SYSTEM Test_10 (* System Configuration *)
  (* Standard: 61499-1 *)
  (* Version 0.3, 2003-12-05, JHC, Rockwell Automation, Renamed from NEWSYSTEM. *)
  (* Version 0.2, 2002-11-05, JHC, Rockwell Automation, Fixed missing (empty) FBD in Application. *)
  (* Version 0.1, 2002-01-17, JHC, Rockwell Automation, Minor cleanup *)
  (* Version 0.0, 2000-05-27, JHC, Rockwell Automation *)
  APPLICATION APP1
  END_APPLICATION
  DEVICE HMI : FRAME_DEVICE(BOUNDS := [500,300,700,500], GRID := [1,1])
    RESOURCE Worker1 : PANEL_RESOURCE(ROWS := 4, COLS := 2)
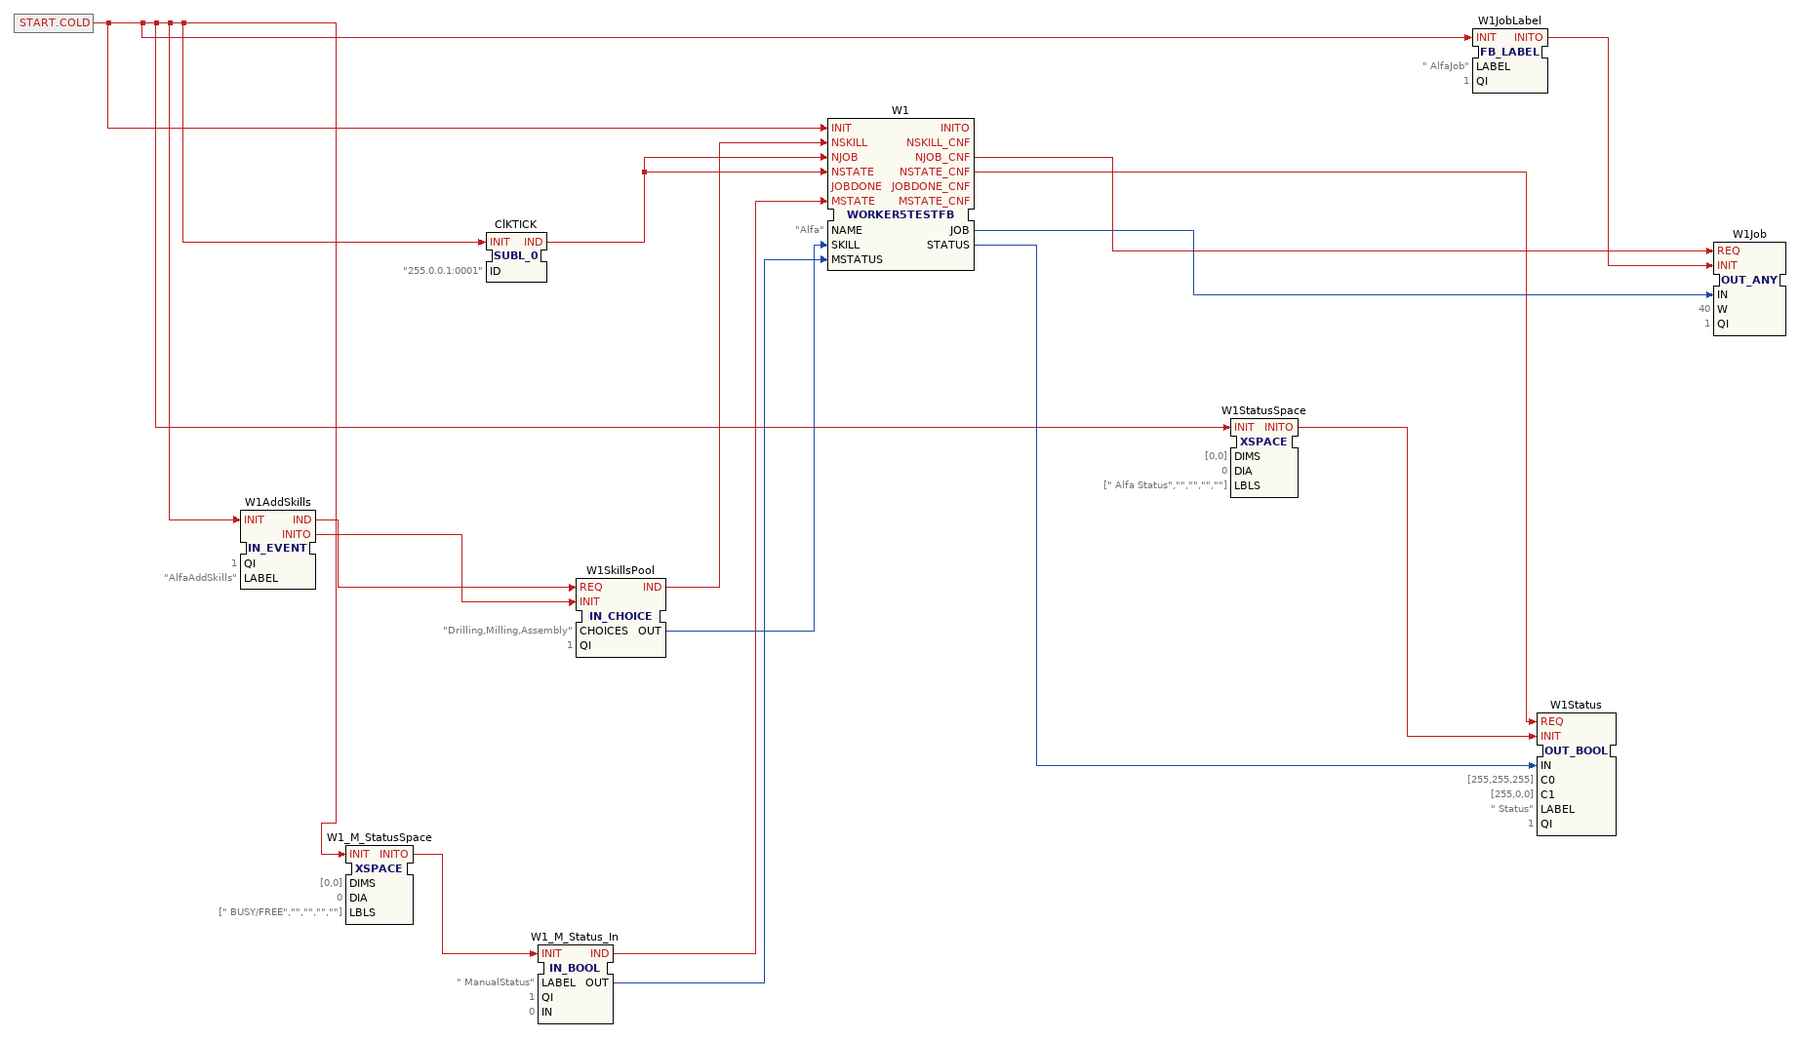
      FBS
        W1 : WORKER5TESTFB(NAME := "Alfa");
        W1SkillsPool : IN_CHOICE(CHOICES := "Drilling,Milling,Assembly", QI := 1);
        W1AddSkills : IN_EVENT(QI := 1, LABEL := "AlfaAddSkills");
        W1Status : OUT_BOOL(C0 := [255,255,255], C1 := [255,0,0], LABEL := "        Status", QI := 1);
        W1Job : OUT_ANY(W := 40, QI := 1);
        W1JobLabel : FB_LABEL(LABEL := "        AlfaJob", QI := 1);
        W1StatusSpace : XSPACE(DIMS := [0,0], DIA := 0, LBLS := ["        Alfa Status","","","",""]);
        ClKTICK : SUBL_0(ID := "255.0.0.1:0001");
        W1_M_Status_In : IN_BOOL(LABEL := "        ManualStatus", QI := 1, IN := 0);
        W1_M_StatusSpace : XSPACE(DIMS := [0,0], DIA := 0, LBLS := ["        BUSY/FREE","","","",""]);
      END_FBS
      EVENT_CONNECTIONS
        START.COLD TO W1.INIT;
        W1SkillsPool.IND TO W1.NSKILL;
        W1AddSkills.IND TO W1SkillsPool.REQ;
        W1.NSTATE_CNF TO W1Status.REQ;
        W1.NJOB_CNF TO W1Job.REQ;
        START.COLD TO W1JobLabel.INIT;
        W1JobLabel.INITO TO W1Job.INIT;
        START.COLD TO W1StatusSpace.INIT;
        W1StatusSpace.INITO TO W1Status.INIT;
        START.COLD TO W1AddSkills.INIT;
        W1AddSkills.INITO TO W1SkillsPool.INIT;
        START.COLD TO ClKTICK.INIT;
        ClKTICK.IND TO W1.NJOB;
        ClKTICK.IND TO W1.NSTATE;
        W1_M_Status_In.IND TO W1.MSTATE;
        START.COLD TO W1_M_StatusSpace.INIT;
        W1_M_StatusSpace.INITO TO W1_M_Status_In.INIT;
      END_CONNECTIONS
      DATA_CONNECTIONS
        W1SkillsPool.OUT TO W1.SKILL;
        W1.JOB TO W1Job.IN;
        W1.STATUS TO W1Status.IN;
        W1_M_Status_In.OUT TO W1.MSTATUS;
      END_CONNECTIONS
    END_RESOURCE
    RESOURCE Worker2 : PANEL_RESOURCE(ROWS := 4, COLS := 2)
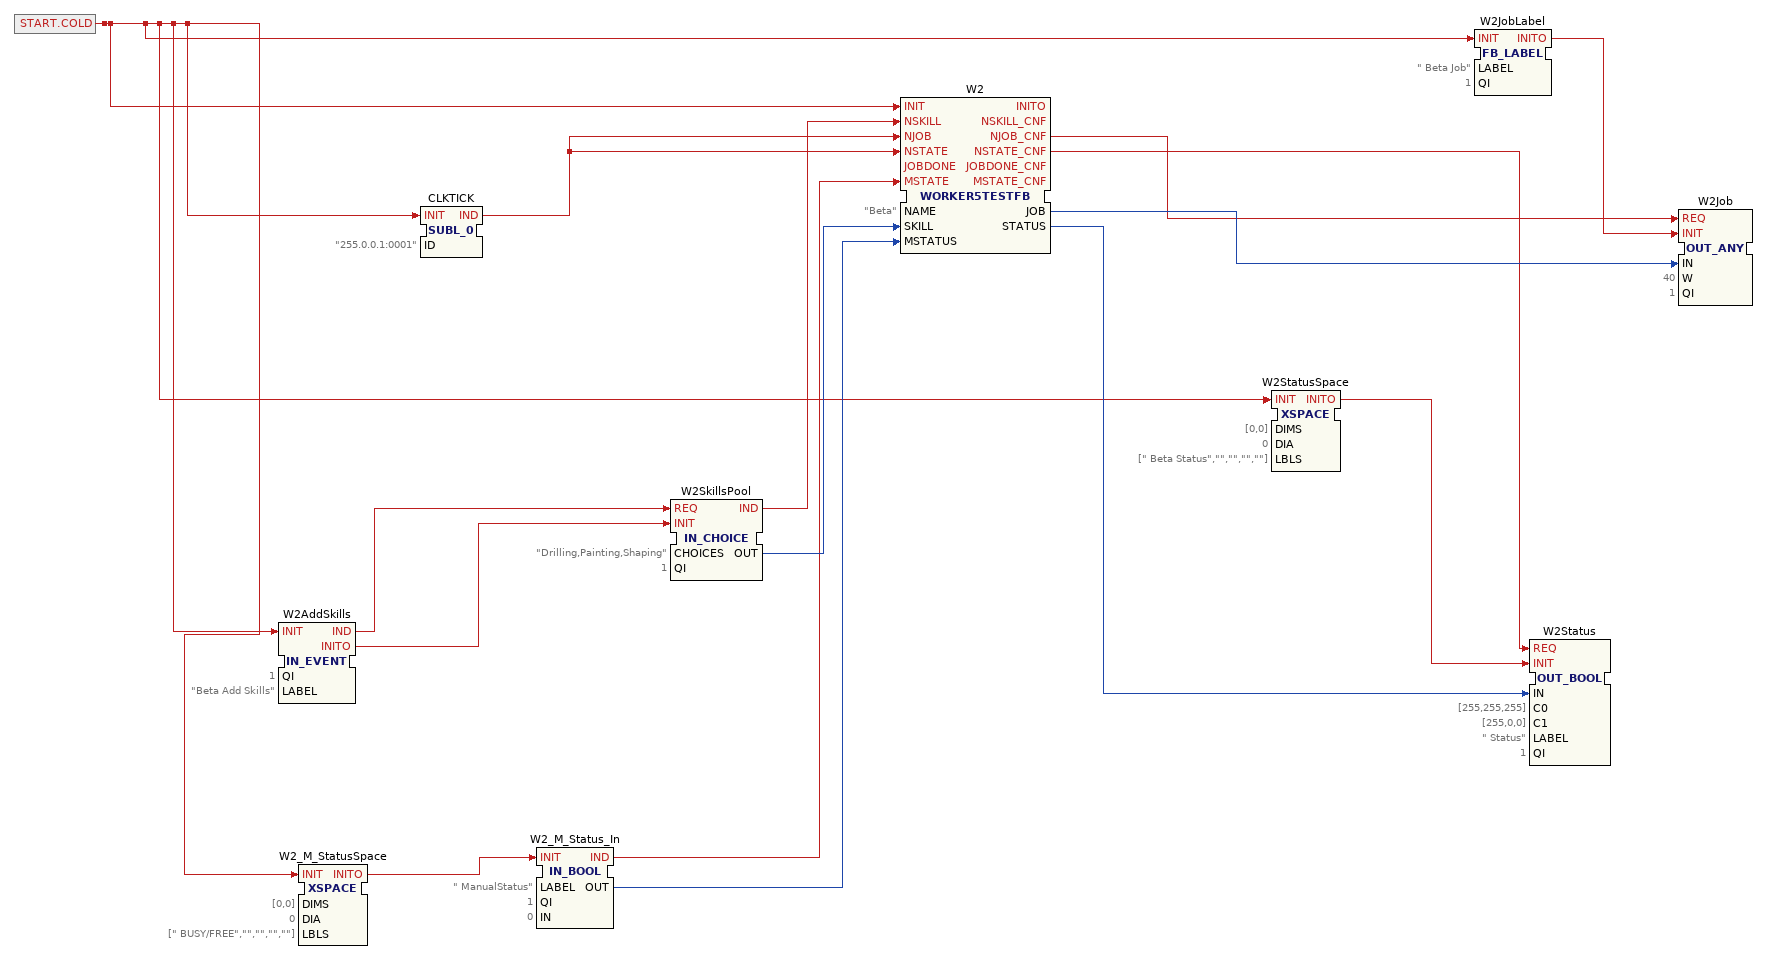
      FBS
        W2 : WORKER5TESTFB(NAME := "Beta");
        W2SkillsPool : IN_CHOICE(CHOICES := "Drilling,Painting,Shaping", QI := 1);
        W2AddSkills : IN_EVENT(QI := 1, LABEL := "Beta Add Skills");
        W2Status : OUT_BOOL(C0 := [255,255,255], C1 := [255,0,0], LABEL := "        Status", QI := 1);
        W2Job : OUT_ANY(W := 40, QI := 1);
        W2JobLabel : FB_LABEL(LABEL := "        Beta Job", QI := 1);
        W2StatusSpace : XSPACE(DIMS := [0,0], DIA := 0, LBLS := ["        Beta Status","","","",""]);
        CLKTICK : SUBL_0(ID := "255.0.0.1:0001");
        W2_M_Status_In : IN_BOOL(LABEL := "      ManualStatus", QI := 1, IN := 0);
        W2_M_StatusSpace : XSPACE(DIMS := [0,0], DIA := 0, LBLS := ["        BUSY/FREE","","","",""]);
      END_FBS
      EVENT_CONNECTIONS
        START.COLD TO W2.INIT;
        W2SkillsPool.IND TO W2.NSKILL;
        W2AddSkills.IND TO W2SkillsPool.REQ;
        W2.NSTATE_CNF TO W2Status.REQ;
        W2.NJOB_CNF TO W2Job.REQ;
        START.COLD TO W2JobLabel.INIT;
        W2JobLabel.INITO TO W2Job.INIT;
        START.COLD TO W2StatusSpace.INIT;
        W2StatusSpace.INITO TO W2Status.INIT;
        START.COLD TO W2AddSkills.INIT;
        W2AddSkills.INITO TO W2SkillsPool.INIT;
        START.COLD TO CLKTICK.INIT;
        CLKTICK.IND TO W2.NJOB;
        CLKTICK.IND TO W2.NSTATE;
        START.COLD TO W2_M_StatusSpace.INIT;
        W2_M_StatusSpace.INITO TO W2_M_Status_In.INIT;
        W2_M_Status_In.IND TO W2.MSTATE;
      END_CONNECTIONS
      DATA_CONNECTIONS
        W2SkillsPool.OUT TO W2.SKILL;
        W2.JOB TO W2Job.IN;
        W2.STATUS TO W2Status.IN;
        W2_M_Status_In.OUT TO W2.MSTATUS;
      END_CONNECTIONS
    END_RESOURCE
  END_DEVICE
  DEVICE Control : FRAME_DEVICE(BOUNDS := [800,800,150,150], GRID := [1,1])
    RESOURCE GlobalClock : PANEL_RESOURCE(ROWS := 0, COLS := 0)
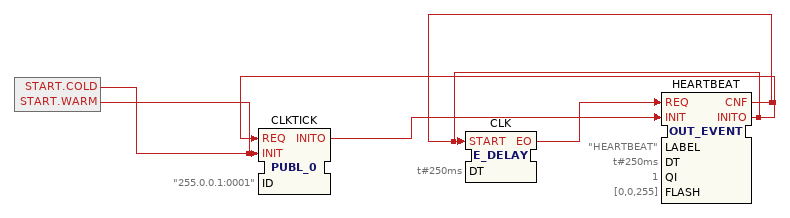
      FBS
        CLKTICK : PUBL_0(ID := "255.0.0.1:0001");
        HEARTBEAT : OUT_EVENT(LABEL := "HEARTBEAT", DT := t#250ms, QI := 1, FLASH := [0,0,255]);
        CLK : E_DELAY(DT := t#250ms);
      END_FBS
      EVENT_CONNECTIONS
        CLK.EO TO HEARTBEAT.REQ;
        HEARTBEAT.CNF TO CLK.START;
        HEARTBEAT.CNF TO CLKTICK.REQ;
        START.COLD TO CLKTICK.INIT;
        START.WARM TO CLKTICK.INIT;
        CLKTICK.INITO TO HEARTBEAT.INIT;
        HEARTBEAT.INITO TO CLK.START;
        HEARTBEAT.INITO TO CLKTICK.REQ;
      END_CONNECTIONS
    END_RESOURCE
  END_DEVICE
  DEVICE Robot : FRAME_DEVICE(GRID := [1,1], BOUNDS := [1200,300,200,200])
    RESOURCE Robot : PANEL_RESOURCE
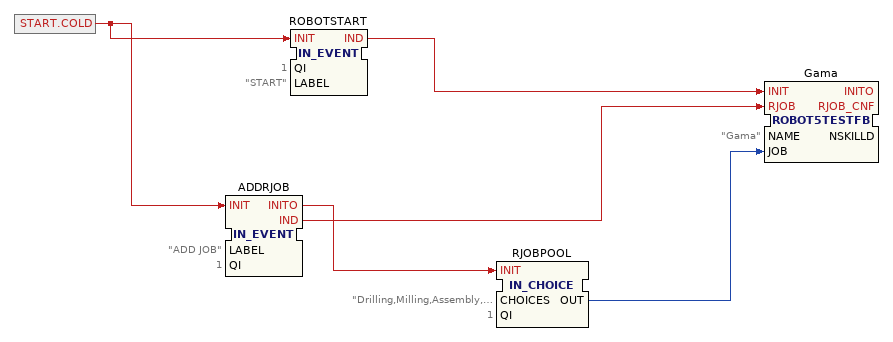
      FBS
        Gama : ROBOT5TESTFB(NAME := "Gama");
        ROBOTSTART : IN_EVENT(QI := 1, LABEL := "START");
        ADDRJOB : IN_EVENT(LABEL := "ADD JOB", QI := 1);
        RJOBPOOL : IN_CHOICE(CHOICES := "Drilling,Milling,Assembly,Painting,Shaping", QI := 1);
      END_FBS
      EVENT_CONNECTIONS
        START.COLD TO ROBOTSTART.INIT;
        ROBOTSTART.IND TO Gama.INIT;
        ADDRJOB.INITO TO RJOBPOOL.INIT;
        START.COLD TO ADDRJOB.INIT;
        ADDRJOB.IND TO Gama.RJOB;
      END_CONNECTIONS
      DATA_CONNECTIONS
        RJOBPOOL.OUT TO Gama.JOB;
      END_CONNECTIONS
    END_RESOURCE
  END_DEVICE
END_SYSTEM
